// TwinCAT 3 PLC project Learning_TwinCat
// ProgramVersion: 3.1.4024.0
// libraries:
//   Tc2_Standard, * (Beckhoff Automation GmbH)
//   Tc2_System, * (Beckhoff Automation GmbH)
//   Tc2_Utilities, * (Beckhoff Automation GmbH)
//   Tc3_Module, * (Beckhoff Automation GmbH)
// project tree:
//   DUTs/ E_EventType.TcDUT (not stored), ST_Events.TcDUT
//   / PlcTask.TcTTO (not stored)
//   POUs/ EvetLogger.TcPOU (not stored), FUpdateEventTimeStampedWithSystemTimeStamepd.TcPOU (not stored), MAIN.TcPOU (not stored)
// real-time tasks:
//   TASK PlcTask: cycle T#10ms, priority 20, ADS port 350

// ---- DUTs/ST_Events.TcDUT
TYPE ST_Events :
STRUCT
	eEventType : E_EventType;
	eEventSeverity : TcEventSeverity;
	eEventIdentity : UDINT;
	eEventText : STRING(255);
	dtTimeStamped : DATE_AND_TIME ;
	
	
END_STRUCT
END_TYPE
